{attribute 'qualified_only'}
VAR_GLOBAL
	bResetFaults		: BOOL 	:= FALSE	; // Reset system faults 
	bCmdSnoozeMessage	: BOOL 	:= FALSE	; // Snooze message display
	bHideFaults			: BOOL 	:= FALSE 	; // Display fault message popup on screen (when MC, CF of FF are active)
	bHideReset			: BOOL 	:= False 	; // Hide reset button in display unless CF of FF is active 
	arActiveFaults 		: ARRAY [0..Param_Messages.nMAX_MESSAGES_SHOWN] OF UDT_Fault ; // Active faults overview for showing in HMI
	sOPeratorMessage	: STRING ;	// operator message for displaying non vital machine data
END_VAR
VAR_GLOBAL CONSTANT 
	tMESSAGESNOOZEDURATION	: TIME 	:= T#5s ; // duration of message snooze after button press 
END_VAR

(* stored: Version 1.1.0.1, ProductVersion 3.1.4024.5
   GVL GVL_Message: Id {50f467a8-facb-42cb-96fd-d0c9df172a76} *)
